Fanuc KAREL source: kb00020.KL

-- PROVISIONAL review KL for V940-1; original PC SHA256 585e33b936e1a779582fb1b71f9b6536fd15ae80cdb140b1c0daf2c1cd16d553
-- Incomplete behavior may be omitted. Consult companion uncertainty JSON. Do not deploy.
PROGRAM KB00020
%NOLOCKGROUP
VAR
  P1 : INTEGER
  RESULT : STRING[80]
BEGIN
  -- V9_ZERO_TABLE_METADATA_HINT layout=0001; no indexed target words; source/name/runtime held
  -- UNRESOLVED_PC offsets 5-12; opcodes 9D,23
  -- UNRESOLVED_PC offsets 17-32; opcodes 27,22,76,75
  -- UNRESOLVED_PC offsets 37-41; opcodes 7F
END KB00020
